Fanuc KAREL source: CHECK_EPOS.kl

PROGRAM T
%NOLOCKGROUP
VAR
 v0 : XYZWPREXT
 v1 : POSITION
 v2 : POSITION
 v3 : INTEGER
 v4 : INTEGER
BEGIN
 CHECK_EPOS(v0, v1, v2, v3, v4)
END T
